INTERFACE I_SysModules

METHOD accept
VAR_INPUT
	iVisitor : I_Visitor;
END_VAR
END_METHOD

END_INTERFACE

(* stored: Version 1.1.0.1, ProductVersion 3.1.4024.12
   Itf I_SysModules: Id {073f48fb-e2af-4b1a-a74f-362700c31e24}
   Method accept: Id {506d095f-0bbc-48c7-a516-c48bc525fbd6} *)
